// TwinCAT 3 PLC project Main
// ProgramVersion: 3.1.4024.0
// libraries:
//   Tc2_Standard, * (Beckhoff Automation GmbH)
//   Tc2_System, * (Beckhoff Automation GmbH)
//   Tc3_Module, * (Beckhoff Automation GmbH)
// project tree:
//   GVLs/ GVL1.TcGVL
//   / PlcTask.TcTTO
//   POUs/ MAIN.TcPOU
// real-time tasks:
//   TASK PlcTask: cycle T#10ms, priority 20, ADS port 350

CONFIGURATION Main
    RESOURCE PLC ON TwinCAT3
        TASK PlcTask(INTERVAL := T#10ms, PRIORITY := 20);
        PROGRAM MAIN WITH PlcTask : MAIN;
    END_RESOURCE
END_CONFIGURATION

// ---- GVLs/GVL1.TcGVL
{attribute 'qualified_only'}
VAR_GLOBAL
	//bemenetek
	i_ajelenlet : ARRAY[0..10] OF	BOOL; //jelenlet
	i_afelhivas : ARRAY[1..9] OF 	BOOL; // hivas fel (0 alatt és 10 fölött mar nincs ezert őket nem vesszük bele)
	i_alehivas : ARRAY[1..9] OF 	BOOL; //hivas le
	i_afulke : ARRAY[0..10] OF 		BOOL; //fülke gombjai
	i_bzartajto AT %I* : 			BOOL; //zart ajto
	i_bnyitottajto AT %I* :			BOOL; //nyitott ajtó
	
	//kimenetek
	q_bfelfele AT %I* : 			BOOL; //felfelé megy
	q_blefele AT %I* :				BOOL; //lefelé megy
	q_anyugtalampa : ARRAY[0..10]OF BOOL; //szintenkénti nyugtázó lámpa
	q_bajtonyit AT %I* :			BOOL; //ajtonyitás
	q_bajtozar AT %I* :				BOOL; //ajtozarva
	q_afulkecelallomsa : ARRAY[0..10] OF BOOL; //fülkeben celallomas
	
	v_ijelenlegi : 					INT ; //jelenlegi emelet
	v_acelallomas : ARRAY[0..10]OF  BOOL; //célállomás
	
	v_tido : 						TON;  // Időzito
	c_tvarakozasiido : TIME := 		T#10S; // Váarakozási idő
			
	
	
END_VAR

// ---- POUs/MAIN.TcPOU
PROGRAM MAIN
VAR
	i: INT := 1;
	
END_VAR

 //emelet
FOR i := 0 TO 10 DO
	IF	GVL1.i_ajelenlet[i] THEN
			GVL1.v_ijelenlegi := i;
	END_IF;
END_FOR;

//megérkezés
IF GVL1.v_acelallomas[GVL1.v_ijelenlegi] THEN 
	GVL1.q_bfelfele := FALSE;
	GVL1.q_blefele := FALSE;
END_IF;

//hívásregisztrálás
FOR i := 0 TO 10 DO
	IF GVL1.i_afelhivas[i] THEN
		GVL1.v_acelallomas[i] := TRUE;
		GVL1.q_anyugtalampa[i] := TRUE; //A lifthívás nyugtázva lett, ennek visszajelzése
	END_IF;
	IF GVL1.i_alehivas[i] THEN
		GVL1.v_acelallomas[i] := TRUE;
		GVL1.q_anyugtalampa[i] := TRUE;
	END_IF;
END_FOR;

//Fülkéből
FOR i := 0 TO 10 DO
	IF GVL1.i_afulke[i] THEN
		GVL1.v_acelallomas[i] := TRUE; // A célemelet beállítása a liftből
		GVL1.q_afulkecelallomsa[i] := TRUE; //fulke lampa 
	END_IF;
END_FOR;

//ajtonyitas
IF GVL1.v_acelallomas[GVL1.v_ijelenlegi] AND NOT GVL1.v_tido.IN THEN // HA célallomason vagyunk és még nem indult az ora
	 	GVL1.i_bnyitottajto := TRUE; 
		GVL1.i_bzartajto := FALSE; // csak nyitott ajtonal
		GVL1.v_tido(IN := TRUE, PT := GVL1.c_tvarakozasiido);	
END_IF;

IF GVL1.v_tido.Q THEN
	GVL1.i_bnyitottajto := FALSE;
	GVL1.i_bzartajto := TRUE;
	GVL1.v_acelallomas[GVL1.v_ijelenlegi] := FALSE;
END_IF;

//Mozgatas
IF NOT GVL1.v_acelallomas[GVL1.v_ijelenlegi] THEN
	FOR i := 0 TO 10 DO
		IF GVL1.v_acelallomas[i] THEN
			IF i < GVL1.v_ijelenlegi THEN // HA a celpont alacsonyabban van mint a lift
				GVL1.q_blefele := TRUE; // A lift lefele megy 
			END_IF;
			IF i > GVL1.v_ijelenlegi THEN // HA a celpont fentebb van mint a lift
				GVL1.q_bfelfele := TRUE; // A lift felfele megy
			END_IF;			
		END_IF;
	END_FOR;
END_IF;

END_PROGRAM
